// Mitsubishi GX Works2 project: 오전터치   PLC: Q03UDV

PROGRAM MAIN
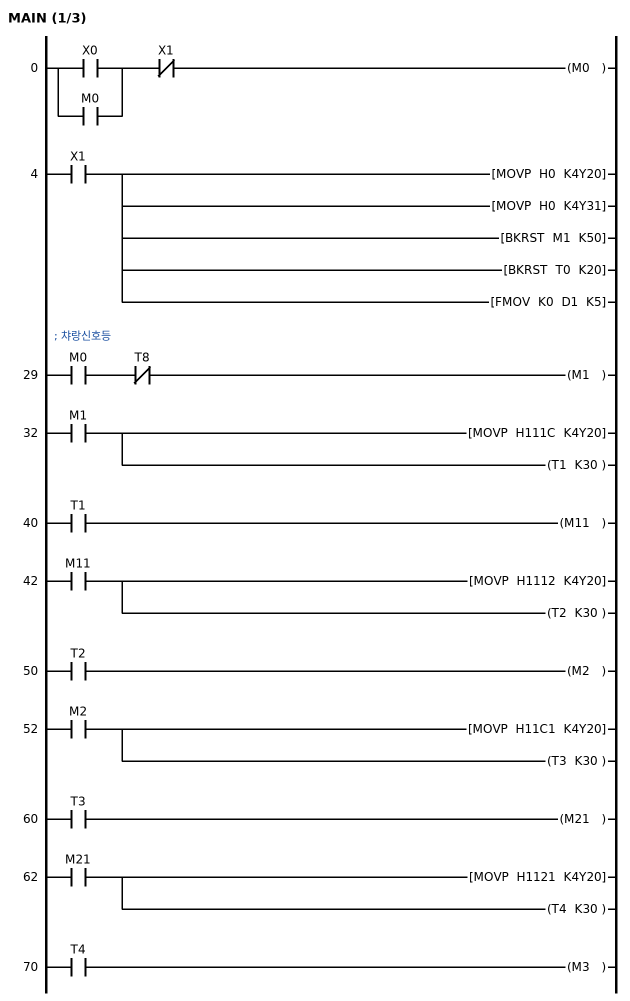
0     LD      X0
      OR      M0
      ANI     X1
      OUT     M0
4     LD      X1
      MOVP    H0 K4Y20
      MOVP    H0 K4Y31
      BKRST   M1 K50
      BKRST   T0 K20
      FMOV    K0 D1 K5
; 챠랑신호등
29    LD      M0
      ANI     T8
      OUT     M1
32    LD      M1
      MOVP    H111C K4Y20
      OUT     T1 K30
40    LD      T1
      OUT     M11
42    LD      M11
      MOVP    H1112 K4Y20
      OUT     T2 K30
50    LD      T2
      OUT     M2
52    LD      M2
      MOVP    H11C1 K4Y20
      OUT     T3 K30
60    LD      T3
      OUT     M21
62    LD      M21
      MOVP    H1121 K4Y20
      OUT     T4 K30
70    LD      T4
      OUT     M3
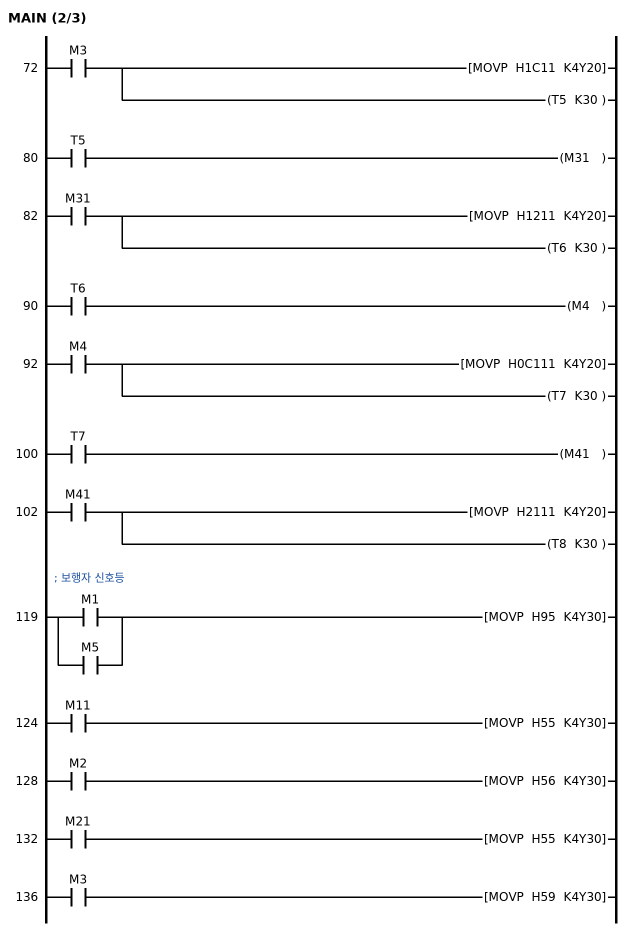
72    LD      M3
      MOVP    H1C11 K4Y20
      OUT     T5 K30
80    LD      T5
      OUT     M31
82    LD      M31
      MOVP    H1211 K4Y20
      OUT     T6 K30
90    LD      T6
      OUT     M4
92    LD      M4
      MOVP    H0C111 K4Y20
      OUT     T7 K30
100   LD      T7
      OUT     M41
102   LD      M41
      MOVP    H2111 K4Y20
      OUT     T8 K30
; 보행자 신호등
119   LD      M1
      OR      M5
      MOVP    H95 K4Y30
124   LD      M11
      MOVP    H55 K4Y30
128   LD      M2
      MOVP    H56 K4Y30
132   LD      M21
      MOVP    H55 K4Y30
136   LD      M3
      MOVP    H59 K4Y30
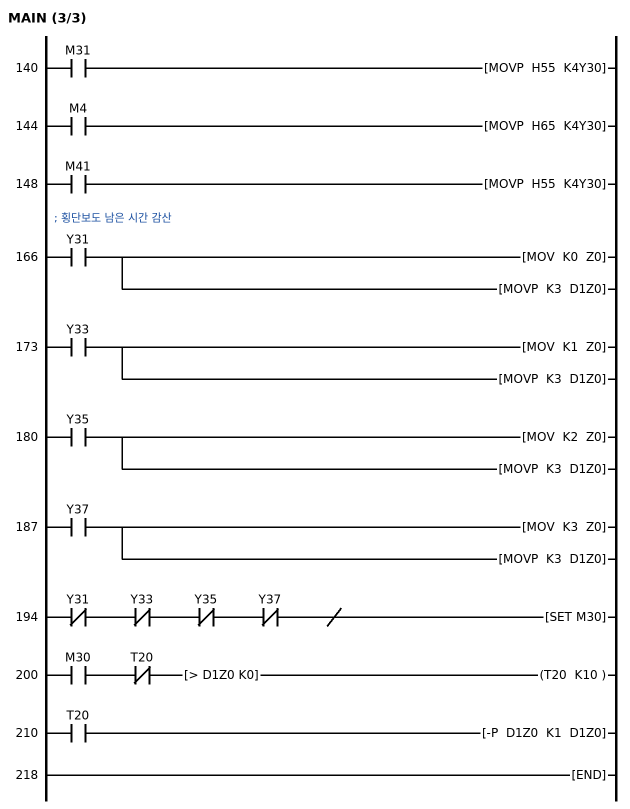
140   LD      M31
      MOVP    H55 K4Y30
144   LD      M4
      MOVP    H65 K4Y30
148   LD      M41
      MOVP    H55 K4Y30
; 횡단보도 남은 시간 감산
166   LD      Y31
      MOV     K0 Z0
      MOVP    K3 D1Z0
173   LD      Y33
      MOV     K1 Z0
      MOVP    K3 D1Z0
180   LD      Y35
      MOV     K2 Z0
      MOVP    K3 D1Z0
187   LD      Y37
      MOV     K3 Z0
      MOVP    K3 D1Z0
194   LDI     Y31
      ANI     Y33
      ANI     Y35
      ANI     Y37
      INV
      SET     M30
200   LD      M30
      ANI     T20
      AND>    D1Z0 K0
      OUT     T20 K10
210   LD      T20
      -P      D1Z0 K1 D1Z0
218   END
END_PROGRAM
